FUNCTION_BLOCK FB_HMI
VAR_INPUT
END_VAR
VAR_OUTPUT
END_VAR
VAR
END_VAR

VAR_IN_OUT
	ST_In			: 	ST_CSL_In;
	ST_Out			:	ST_CSL_Out;
	ST_Page			:	ST_HMI_Page;
	ST_DisplayName	:	ST_HMI_DisplayName;
	ST_Enable		:	ST_HMI_Enable;
	ST_Params		:	ST_CSL_Params;
END_VAR


IF ST_Page.Numbers_page = 0  THEN
	
	ST_Page.Home_page := TRUE;
	ST_Page.Allarms_page := FALSE;
	ST_Page.Params_page := FALSE;
	
END_IF

IF ST_Page.Numbers_page = 1  THEN
	
	ST_Page.Home_page := FALSE;
	ST_Page.Allarms_page := TRUE;
	ST_Page.Params_page := FALSE;
	
END_IF

IF ST_Page.Numbers_page = 2  THEN
	
	ST_Page.Home_page := FALSE;
	ST_Page.Allarms_page := FALSE;
	ST_Page.Params_page := TRUE;
	
END_IF

IF ST_Enable.ClosePopUp = TRUE	THEN
	
	ST_Enable.GeneralEnable	:= FALSE;
	
END_IF

IF ST_Enable.Valve1 = TRUE	THEN
	
	ST_Enable.GeneralEnable	:= TRUE;
	ST_DisplayName.DisplayName	:=	ST_DisplayName.Valve1;
	ST_Enable.GeneralState	:= ST_Out.bValveSlot1;
	
END_IF

END_FUNCTION_BLOCK

(* stored: Version 1.1.0.1, ProductVersion 3.1.4024.12
   POU FB_HMI: Id {2a92276f-68aa-42a1-8ada-c02f33716a1b}, SpecialFunc None *)
